(* IEC 61131-3 sources: MotionTestBenchMaster/Logical/00_AID/Libraries/Sidel_Libraries/ITC/UDP_COM, 4 files *)

(* ---- UDP_COM.typ ---- *)
(********************************************************************
 * COPYRIGHT - Sidel Spa
 ********************************************************************
 * Library: UDP_COM
 * File: UDP_COM.typ
 * Author: Andrea.Cortesi
 * Created: May 28, 2013
 ********************************************************************
 * Data types of library UDP_COM
 ********************************************************************)

TYPE
	UDP_DataType : 	STRUCT
		Connection_OK : BOOL;
		Com_Status : UINT; (*(0=Connect OK;1=Not Enabled;2=Error Sending;3=Error Receiving;10=Connection Waiting)*)
	END_STRUCT;
END_TYPE

(* ---- UDP_COM.fun ---- *)
(********************************************************************
 * COPYRIGHT -- Sidel
 ********************************************************************
 * Library: UDP_COM
 * File: UDP_COM.fun
 * Author: Andrea.Cortesi
 * Created: May 28, 2013
 ********************************************************************
 * Functions and function blocks of library UDP_COM
 ********************************************************************)

FUNCTION_BLOCK UDP_COM (*UDP Communication Function*)
	VAR_INPUT
		Enable_Com : BOOL; (*Enable Communication*)
		IP_Address : STRING[40]; (*Partner IP address. (e.g. '10.1.92.20') (as a string)*)
		Local_Port : UINT; (*Local port number.*)
		Remote_Port : UINT; (*Remote port number.*)
		Recv_Buffer : UDINT; (*Received data buffer address (string given as a pointer)*)
		Recv_Length : UDINT; (*Reiceved data maximum length (in bytes)*)
		Send_Buffer : UDINT; (*Data to send buffer address (string given as a pointer)*)
		Send_Length : UDINT; (*Sent data length (in bytes)*)
		Rcv_Time_Out : TIME; (*Reception time out setpoint (in ms) (typical value: 1000ms)*)
		Send_Time_Act : TIME; (*Data send time cadence (in ms) (typical value: 100ms)*)
	END_VAR
	VAR_OUTPUT
		Connection_OK : BOOL; (*True = both PLCs are connected*)
		Recv_Data_Length : UDINT; (*Length of the bytes received.*)
		Send_Data_Length : UDINT; (*Length of the bytes send*)
		Status : USINT; (*Communication status. Status = 0, means communication is OK*)
		Status_Message : STRING[25]; (*Communication status string*)
	END_VAR
	VAR
		Socket_ID : UDINT; (*Identifier sent by the UdpOpen block *)
		UDP_Com_UdpOpen : UdpOpen; (*Communication opening function block*)
		UDP_Com_UdpClose : UdpClose; (*Communication closing function block*)
		UDP_Com_UdpSend : UdpSend; (*Data sending function block*)
		UDP_Com_UdpRecv : UdpRecv; (*Data receiving function block*)
		UDP_Step : USINT; (*Implemented communication block status*)
		Open_Status : UINT; (*Communication opening function block status*)
		Send_Status : UINT; (*Data sending function block status*)
		Recv_Status : UINT; (*Data receiving function block status*)
		Close_Status : UINT; (*communication closing function block status*)
		Send_Timer : TON; (*Sending timer*)
		Rcv_Timer : TON; (*Receiveing timer*)
		ConnectTimeOut_Timer : TON; (*Connection Time Out*)
	END_VAR
END_FUNCTION_BLOCK

(* ---- UDP_COM.st ---- *)
(********************************************************************
 * COPYRIGHT -- Sidel
 ********************************************************************
 * Library: UDP_COM
 * File: UDP_COM.st
 * Author: Andrea.Cortesi
 * Created: Jun 26, 2013
 ********************************************************************
 * Implementation of library UDP_COM
 ********************************************************************)

(* UDP COMMUNICATION FUNCTION BLOC IMPLEMENTATION *)
FUNCTION_BLOCK UDP_COM

	Send_Timer.PT := Send_Time_Act;
	Send_Timer();

	Rcv_Timer.PT := Rcv_Time_Out;
	Rcv_Timer();

	ConnectTimeOut_Timer.PT := T#2000ms;
	ConnectTimeOut_Timer();

	IF Rcv_Timer.Q THEN
		(* Close Communication UDP *)
		UDP_Step := 60;
	END_IF

	CASE UDP_Step OF

		0:	(* Open UDP Connection *)

			Rcv_Timer.IN := FALSE;

			IF Enable_Com THEN
				Status := UDP_Connection_Waiting;
			ELSE
				Status := UDP_Not_Enabled;
			END_IF

			UDP_Com_UdpOpen.enable	 := Enable_Com;
			UDP_Com_UdpOpen.pIfAddr  := 0;           (* Listen on all UDP Interfaces*)
			UDP_Com_UdpOpen.port 	 := Local_Port;  (* Port to listen*)
			UDP_Com_UdpOpen.options  := udpOPT_REUSEADDR;

			UDP_Com_UdpOpen();    (* Call the Function*)

			Socket_ID 	             := UDP_Com_UdpOpen.ident;
			Open_Status              := UDP_Com_UdpOpen.status;

			IF Open_Status = 0 THEN  (* UdpOpen successful*)
				(* Initialization Send and Receive Ident *)
				UDP_Step := 40;
			END_IF

			Connection_OK := FALSE;

		40: (* Initialization Send and Receive Ident *)

			Rcv_Timer.IN := TRUE;

			(* Data send block parameters *)
			UDP_Com_UdpSend.enable  := TRUE;
			UDP_Com_UdpSend.ident   := Socket_ID;	                    (* Client Ident from UDP_Open *)
			UDP_Com_UdpSend.pHost   := ADR(IP_Address);	                (* IP Address of remote partner *)
			UDP_Com_UdpSend.port    := Remote_Port;		                (* Port number of remote partner *)
			UDP_Com_UdpSend.pData   := Send_Buffer;	                    (* Which data to send *)
			UDP_Com_UdpSend.datalen := Send_Length;	                    (* Lenght of data to send *)
			UDP_Com_UdpSend.flags   := 0;

			(* Data receive block parameters *)
			UDP_Com_UdpRecv.enable  := TRUE;
			UDP_Com_UdpRecv.ident   := Socket_ID;	                    (* Client Ident from UDP_Open *)
			UDP_Com_UdpRecv.pIpAddr := ADR(IP_Address);	                (* IP Address of remote partner *)
			UDP_Com_UdpRecv.pData   := Recv_Buffer;	                    (* Where to store the incoming data *)
			UDP_Com_UdpRecv.datamax := Recv_Length;                     (* Lenght of data buffer *)
			UDP_Com_UdpRecv.flags   := 0;

			UDP_Step := 50;

			IF NOT(Enable_Com) THEN
				UDP_Step := 0;
			END_IF

			Connection_OK := FALSE;

		50: (* Send and Receive Data *)

			Send_Timer.IN := NOT(Send_Timer.Q);

			UDP_Com_UdpRecv();  (* Call the "Data Recv" function block *)

			Recv_Status        := UDP_Com_UdpRecv.status;
			Recv_Data_Length   := UDP_Com_UdpRecv.recvlen;

			IF Send_Timer.Q THEN
				UDP_Com_UdpSend.enable := TRUE;
			END_IF

			UDP_Com_UdpSend();	(* Call the "Data Sent" function block *)

			Send_Status        := UDP_Com_UdpSend.status;
			Send_Data_Length   := UDP_Com_UdpSend.sentlen;
			Status 	 	       := UDP_Connected_OK;

			IF UDP_Com_UdpSend.enable THEN

				IF (Send_Status <> 65535) AND (Send_Status <> 0) THEN
					UDP_Step := 60;
					Status   := UDP_Error_Sending;
				END_IF

				IF (Send_Status = 0) THEN
					Send_Timer.IN := FALSE;
				ELSE
					Send_Timer.IN := TRUE;
				END_IF

			END_IF

			IF (Recv_Status <> 65535) AND (Recv_Status <> 0) AND (Recv_Status <> udpERR_NO_DATA) THEN
				UDP_Step := 60;
				Status   := UDP_Error_Receiving;
			END_IF

			IF (Recv_Status = 0) THEN
				Rcv_Timer.IN := FALSE;
			ELSE
				Rcv_Timer.IN := TRUE;
			END_IF

			IF NOT(Enable_Com) THEN
				UDP_Step := 60;
			END_IF

			Connection_OK := TRUE;

		60: (* Close Communication UDP *)

			Rcv_Timer.IN := FALSE;

			UDP_Com_UdpClose.enable := TRUE;
			UDP_Com_UdpClose.ident  := Socket_ID;
			UDP_Com_UdpClose();

			Close_Status := UDP_Com_UdpClose.status;
			Status 	 	 := UDP_Connection_Close;

			IF (Close_Status = 0) THEN
				UDP_Step := 70;
			END_IF

			Connection_OK := FALSE;

		70: (* Wait Open New Connection *)

			Rcv_Timer.IN            := FALSE;
			ConnectTimeOut_Timer.IN := TRUE;

			IF ConnectTimeOut_Timer.Q THEN
				UDP_Step                := 0;
				ConnectTimeOut_Timer.IN := FALSE;
			END_IF

			Status 	 	  := UDP_Connection_Waiting;
			Connection_OK := FALSE;

		ELSE

			UDP_Step := 60;

	END_CASE

	CASE Status OF

		0: Status_Message := 'UDP Connection OK';
		1: Status_Message := 'UDP Not Enabled';
		2: Status_Message := 'UDP Error Sending';
		3: Status_Message := 'UDP Error Receiving';
		4: Status_Message := 'UDP Connection Close';
		5: Status_Message := 'UDP Send Receive Run';
	   10: Status_Message := 'UDP Connection Waiting';

	ELSE
		   Status_Message := 'Not Define';
	END_CASE

END_FUNCTION_BLOCK

(* ---- UDP_COM.var ---- *)
(********************************************************************
 * COPYRIGHT -- Sidel
 ********************************************************************
 * Library: UDP_COM
 * File: UDP_COM.var
 * Author: Andrea.Cortesi
 * Created: May 28, 2013
 ********************************************************************
 * Constants of library UDP_COM
 ********************************************************************)
VAR CONSTANT
	UDP_Connected_OK : USINT := 0;
	UDP_Not_Enabled : USINT := 1;
	UDP_Error_Sending : USINT := 2;
	UDP_Error_Receiving : USINT := 3;
	UDP_Connection_Close : USINT := 4;
	UDP_Connection_Waiting : USINT := 10;
END_VAR
